// SIMATIC S7-200 project (STEP 7-Micro/WIN), CPU 221 REL 01.10

SYMBOL_TABLE IO
自动/手动            I0.0
急停按钮             I0.1
启动按钮             I0.2
复位按钮             I0.3
流水线顶升气缸下降检测      I1.0
流水线顶升气缸顶升检测      I1.1
自制气缸松开检测         I1.2
自制气缸夹紧检测         I1.3
电动缸SRDY          I2.0
电动缸STOP          I2.1
电动缸ALRM          I2.2
上工位检测            I3.5
本工位检测            I3.6
下工位检测            I3.7
通道0              IW64
通道1              IW66
电动缸上电            Q0.0
电动缸急停            Q0.1
红灯               Q0.4
黄灯               Q0.5
绿灯               Q0.6
蜂鸣器              Q0.7
流水线顶升气缸顶升        Q1.0
流水线顶升气缸下降        Q1.1
上阻挡器放行           Q2.0
本阻挡器放行           Q2.1
自制气缸夹紧           Q2.2
自制气缸松开           Q2.3
END_SYMBOL_TABLE

SYMBOL_TABLE M3000
流水线工步号           MW3000
产品类型             MW3002
RFID工步号          MW3004
芯片编号             MW3006
一键初始化工步号         MW3008
通讯状态             M3010.0
本工位合格            M3010.1
本工位完成            M3010.2
不合格报警            M3010.3
RFID读取触发         M3010.4
RFID读取完成         M3010.5
M一键初始化按钮         M3011.0
M一键初始化完成         M3011.1
M自制气缸松开          M3021.0
M自制气缸夹紧          M3021.1
M上阻挡器放行          M3020.0
M本阻挡器放行          M3020.2
M随行板顶升           M3020.4
M随行板下降           M3020.5
上工位合格            M3030.0
上工位完成            M3030.1
联线状态             M3040.0
报警工步号            MW3050
RFID运行中          M3010.6
员工权限             M3060.0
END_SYMBOL_TABLE
